FUNCTION_BLOCK Carriage
  (* Standard: 61499-2 *)
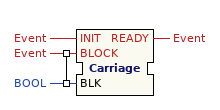
  EVENT_INPUT
    INIT;
    BLOCK WITH BLK;
  END_EVENT
  EVENT_OUTPUT
    READY;
  END_EVENT
  VAR_INPUT
    BLK : BOOL;
  END_VAR
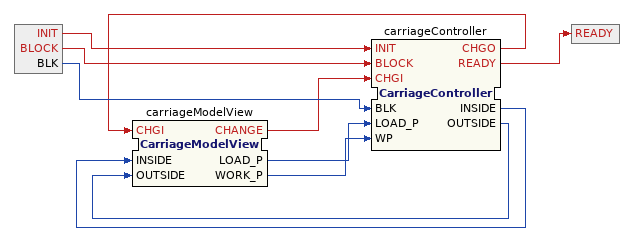
  FBS
    carriageModelView : CarriageModelView;
    carriageController : CarriageController;
  END_FBS
  EVENT_CONNECTIONS
    carriageController.CHGO TO carriageModelView.CHGI;
    carriageController.READY TO READY;
    INIT TO carriageController.INIT;
    BLOCK TO carriageController.BLOCK;
    carriageModelView.CHANGE TO carriageController.CHGI;
  END_CONNECTIONS
  DATA_CONNECTIONS
    BLK TO carriageController.BLK;
    carriageController.INSIDE TO carriageModelView.INSIDE;
    carriageController.OUTSIDE TO carriageModelView.OUTSIDE;
    carriageModelView.LOAD_P TO carriageController.LOAD_P;
    carriageModelView.WORK_P TO carriageController.WP;
  END_CONNECTIONS
END_FUNCTION_BLOCK
